{attribute 'GeneratedUsingTerminal: KL9900-0062'}
{attribute addProperty BoxType "KL9900-0062"}
{attribute addProperty Id "E_StopAT %I*BOOL0"}
{attribute addProperty CRC "1706518016"}
{attribute addProperty Size "0"}
TYPE Channel_65B76600 :
STRUCT
	{attribute addProperty Name "E_Stop"}
	E_Stop AT %I* : BOOL;
END_STRUCT
END_TYPE

(* stored: Version 1.2.0.0, ProductVersion 3.1.4024.9
   DUT Channel_65B76600: Id {f19536c6-1010-46b5-90f7-5b22ccc14d39} *)
